ABB RAPID module: Wobj_FRAME_BufferB.mod

MODULE Wobj_FRAME_BufferB
	! Points are read in order of declaration.
  ! Please do not change the order of points!

  LOCAL PERS robtarget pWobj_U_PointX1:=[[1561.419,601.1981,111.7369],[0.00534455757588148,-0.55362331867218,-0.832725644111633,-0.00637167599052191],[0,0,0,0],[9E+09,9E+09,9E+09,9E+09,9E+09,9E+09]];
	LOCAL PERS robtarget pWobj_U_PointX2:=[[1583.329,-599.8918,111.8258],[0.00534965703263879,-0.55363529920578,-0.832717657089233,-0.00636897888034582],[-1,0,0,0],[9E+09,9E+09,9E+09,9E+09,9E+09,9E+09]];
	LOCAL PERS robtarget pWobj_U_PointY1:=[[2756.826,614.6222,118.7511],[0.00512294936925173,-0.553597509860992,-0.83274245262146,-0.00659863697364926],[0,0,0,0],[9E+09,9E+09,9E+09,9E+09,9E+09,9E+09]];

ENDMODULE
